// TIA Portal V18 export
FUNCTION_BLOCK "BTNS_FB"   // FB1, FBD
{ S7_Optimized_Access := 'TRUE' }
VERSION : 0.1
// stored: AutoNumber true, IsIECCheckEnabled false, IsRetainMemResEnabled false, MemoryReserve 100, SetENOAutomatically false, UDAEnableTagReadback false
   VAR_INPUT
      "remote key activated" : Bool;
      xCylceStart : Bool;
      xDefectMark : Bool;
      xDefectNext : Bool;
      xDefectPrev : Bool;
      xHome : Bool;
      xLaser : Bool;
      xLoad : Bool;
      xControl1 : Bool;
      xControl2 : Bool;
      xbDoorsFwdClose : Bool;
      xbDoorsRevOpen : Bool;
      xbo1Tiltfwd : Bool;
      xbo1Tiltrev : Bool;
      xbo2RotHome : Bool;
      xbo2Rotrev : Bool;
      xSwAuto : Bool;
      xSwMan : Bool;
      xbXfwd : Bool;
      xbxrev : Bool;
      xbyfwd : Bool;
      xbyrev : Bool;
      xbzfwd : Bool;
      xbzrev : Bool;
      xbo2Rotfwd : Bool;
   END_VAR
   VAR_OUTPUT
      remPowerOut : Bool;
      yLedShutter : Bool;
      yLedAuto : Bool;
      ysirenFinished : Bool;
      ySirenError : Bool;
   END_VAR
   VAR
      desk_yledShutter { S7_SetPoint := 'True'} : "LED_FBD";
   END_VAR
   VAR_TEMP   // added for the SCL form of the ladder/FBD networks
      _w1 : Bool;
   END_VAR
BEGIN

REGION Network 2
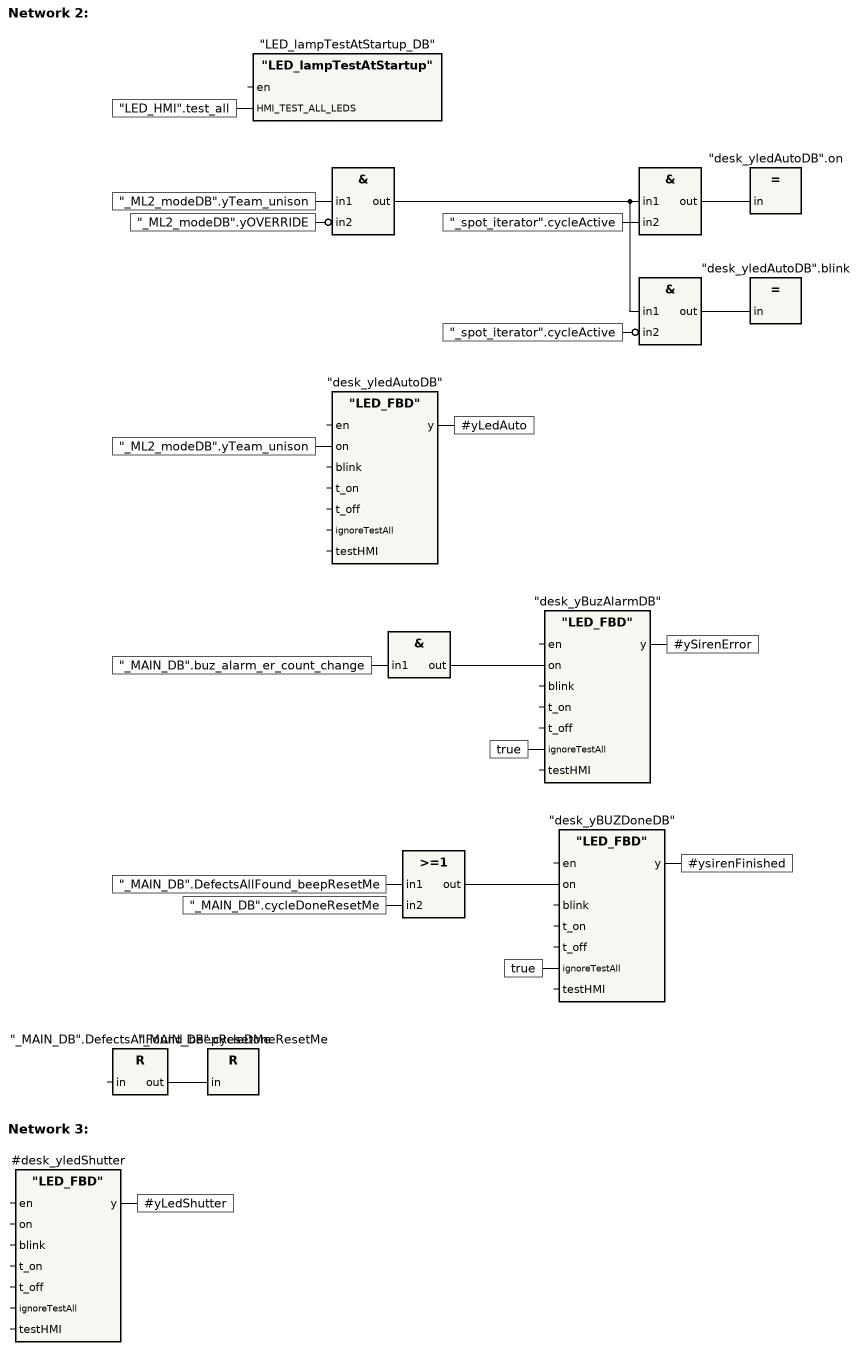
   "LED_lampTestAtStartup_DB"(HMI_TEST_ALL_LEDS := "LED_HMI".test_all);   // "LED_lampTestAtStartup"
   #_w1 := "_ML2_modeDB".yTeam_unison AND NOT "_ML2_modeDB".yOVERRIDE;
   "desk_yledAutoDB".on := #_w1 AND "_spot_iterator".cycleActive;
   "desk_yledAutoDB".blink := #_w1 AND NOT "_spot_iterator".cycleActive;
   "desk_yledAutoDB"(on := "_ML2_modeDB".yTeam_unison, y => #yLedAuto);   // "LED_FBD"
   "desk_yBuzAlarmDB"(on := "_MAIN_DB".buz_alarm_er_count_change, ignoreTestAll := true, y => #ySirenError);   // "LED_FBD"
   "desk_yBUZDoneDB"(on := "_MAIN_DB".DefectsAllFound_beepResetMe OR "_MAIN_DB".cycleDoneResetMe,   // "LED_FBD"
                     ignoreTestAll := true,
                     y => #ysirenFinished);
   "_MAIN_DB".DefectsAllFound_beepResetMe := FALSE;
   "_MAIN_DB".cycleDoneResetMe := FALSE;
END_REGION

REGION Network 3
   #desk_yledShutter(y => #yLedShutter);   // "LED_FBD"
END_REGION

REGION Network 6
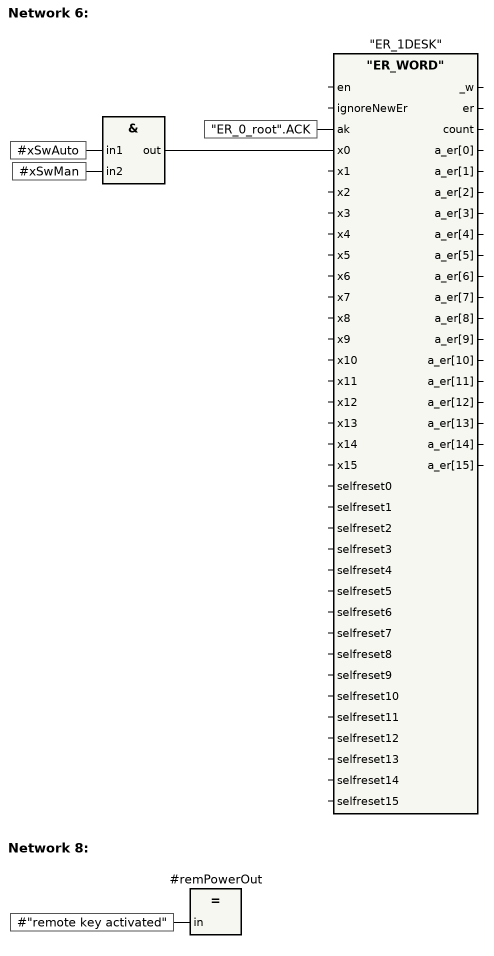
   "ER_1DESK"(ak := "ER_0_root".ACK, x0 := #xSwAuto AND #xSwMan);   // "ER_WORD"
END_REGION

REGION Network 8
   #remPowerOut := #"remote key activated";
END_REGION
END_FUNCTION_BLOCK
